// TIA Portal V20 export
DATA_BLOCK "GDB_Control"   // DB3
TITLE = GDB_Control (minimal)
{ S7_Optimized_Access := 'TRUE' }
// Minimal control DB for ABCDE 5-point cycle. Holds kinematic enable/home arrays + mirror status. Trimmed from v9 (palletizing/recipe/manual fields removed).
// stored: MemoryReserve 100
   VAR
      enableAxes : Bool;   // Enable kinematic group via LKinCtrl_MC_GroupPower
      axesEnabled : Bool;   // Status: all axes enabled (mirror from MC_GroupPower.axesEnabled)
      resetAxes : Bool;   // Reset kinematic group via LKinCtrl_MC_GroupReset
   END_VAR
   VAR RETAIN
      axesError : Bool;   // Status: error on any joint TO
   END_VAR
   VAR
      homeAxes : Bool;   // Home kinematic group via LKinCtrl_MC_GroupHome
      axesHomed : Bool;   // Status: all 4 joint TOs report StatusWord.X5 (Homed)
      axesReady : Bool;   // Phase G (C67, 2026-05-18) — derived: axesEnabled AND axesHomed AND NOT axesError. Computed in FB_AxisCtrl REGION StatusDerived. Per HMI cycle-7.1 BackColor Q2 ACK: single Bool tag enables HMI lmpKinReady_Ubp BackColor Range "1:1" binding without multi-tag JS compute.
      robotStandstill : Bool;   // Status: all 4 joint TOs report StatusWord.X7 (Standstill)
   END_VAR
   VAR RETAIN
      HomePos : Array[1..6] of LReal;   // Home positions per kinematic axis index (A1=J1, A2=J3, A3=J2, A4=J4). Initialized by Startup.scl.
   END_VAR
   VAR
      HomeMode : Array[1..6] of Int;   // Home mode per kinematic axis index. 7 = set actual position (no physical homing motion).
      StartMode : Array[1..6] of DInt;   // Start mode for MC_Power per axis. 1 = enable position-controlled. Initialized by Startup.scl to avoid retain-drift issues.
      StopMode : Array[1..6] of Int;   // Stop mode for MC_Power per axis. 1 = immediate stop. Initialized by Startup.scl.
      RestartMode : Array[1..7] of Bool;   // Restart mode flags for MC_GroupReset per axis.
      bo_gripperGrip : Bool;   // V3.0 (2026-05-19): suction-cup GRIP command (level, TRUE while box attached). Maps to MCD signal `sScaraGrip` (SignalAdapter, Input bool, MCD reads). Driven by FB_AutoCtrl_Palletizing V3.0: latched TRUE from PICK_DESCEND.Done through PLACE_DESCEND.Done; FALSE elsewhere.
      bo_gripperRelease : Bool;   // V3.0 (2026-05-19): suction-cup RELEASE command (pulse, TRUE briefly during active release). Maps to MCD signal `sScaraRelease` (SignalAdapter, Input bool, MCD reads). Driven by FB_AutoCtrl_Palletizing V3.0: pulses TRUE for lr_GripperOpenMs duration after PLACE_DESCEND.Done; FALSE elsewhere. Provides positive box-detach signal beyond just turning off vacuum.
   END_VAR
BEGIN
END_DATA_BLOCK
